PROGRAM Ax06
VAR
	iAxisNumber : INT := E_AxisNames.IncSlits_West;
	iGroupNumber : INT := 3;
	
	stoRTrig : R_Trig;
END_VAR

//Initial parameters of an Axis
IF _TaskInfo[fbGetCurTaskIndex.index].FirstCycle THEN
    //Initial default values:
    GVL.astAxesLocal[iAxisNumber].stHomingConfig.eHomeSeq :=E_HomingRoutines.eHomeToEncPulse_BWD_FAST;
	GVL.astAxesLocal[iAxisNumber].stHomingConfig.fHomeAbsPosition:= -12.5;
	GVL.astAxesLocal[iAxisNumber].stHomingConfig.fHomeMidRelativeMove:=1;
    GVL.astAxesLocal[iAxisNumber].stHomingConfig.fHomePosition := -12.5;
    GVL.astAxesLocal[iAxisNumber].stHomingConfig.fHomeFinishDistance := 0.0;
    GVL.astAxesLocal[iAxisNumber].stConfig.eRestorePosition := E_RestorePosition.eRestoreWithoutHome;
	GVL.astAxesLocal[iAxisNumber].stControl.bAutoEnableDisable := TRUE;
	GVL.astAxesLocal[iAxisNumber].stControl.tMoveFinishedDelay := T#0.1S;
	//Set which group this axis belongs to
	GVL.astAxesLocal[iAxisNumber].stDescription.iGroupNumber := iGroupNumber;
	GVL.astAxesLocal[iAxisNumber].Commissioning := FALSE;
END_IF

//Permit
GVL.astAxesLocal[iAxisNumber].stInputs.bPermit := SAFETY.SAMPLE_PERMIT;

//Safety stop motion
IF SAFETY.STOP_MOTION THEN
	GVL.astAxesLocal[iAxisNumber].stControl.bHalt:= TRUE;
END_IF

stoRTrig(CLK:=GVL.astAxesLocal[iAxisNumber].stStatus.bSTOActive);
IF stoRTrig.Q THEN
	GVL.astAxesLocal[iAxisNumber].stControl.bReset:= TRUE;
END_IF




//Define ACTIONS() or write exclusive code for an specific axis.
(*Eg. Stop when temperature reaches certain values, reduce speed if  a signal is activated, etc.
Eg. GVL.astAxesLocal[x].stControl.bInterlockFwd := NOT bInterlockFwdOK;*)

END_PROGRAM

(* stored: Version 1.1.0.1, ProductVersion 3.1.4026.18
   POU Ax06: Id {82bfc13c-168b-4dfc-8e53-256eef8cedb2}, SpecialFunc None *)
